// Mitsubishi GX Works2 project: Lycoming6p   PLC: FX3U/FX3UC
// AMX-FX3U with EM3A-AM8

PROGRAM MAIN
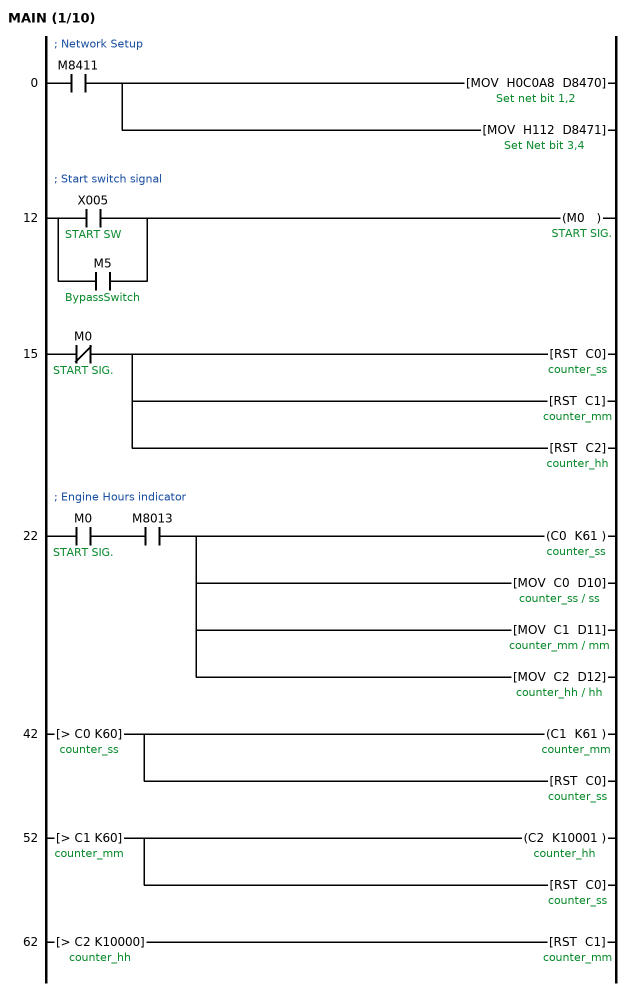
; Network Setup
0     LD      M8411
      MOV     H0C0A8 D8470  ; Set net bit 1,2
      MOV     H112 D8471  ; Set Net bit 3,4
; Start switch signal
12    LD      X005  ; START SW
      OR      M5  ; BypassSwitch
      OUT     M0  ; START SIG.
15    LDI     M0  ; START SIG.
      RST     C0  ; counter_ss
      RST     C1  ; counter_mm
      RST     C2  ; counter_hh
; Engine Hours indicator
22    LD      M0  ; START SIG.
      AND     M8013
      OUT     C0 K61  ; counter_ss
      MOV     C0 D10  ; ss
      MOV     C1 D11  ; mm
      MOV     C2 D12  ; hh
42    LD>     C0 K60  ; counter_ss
      OUT     C1 K61  ; counter_mm
      RST     C0  ; counter_ss
52    LD>     C1 K60  ; counter_mm
      OUT     C2 K10001  ; counter_hh
      RST     C0  ; counter_ss
62    LD>     C2 K10000  ; counter_hh
      RST     C1  ; counter_mm
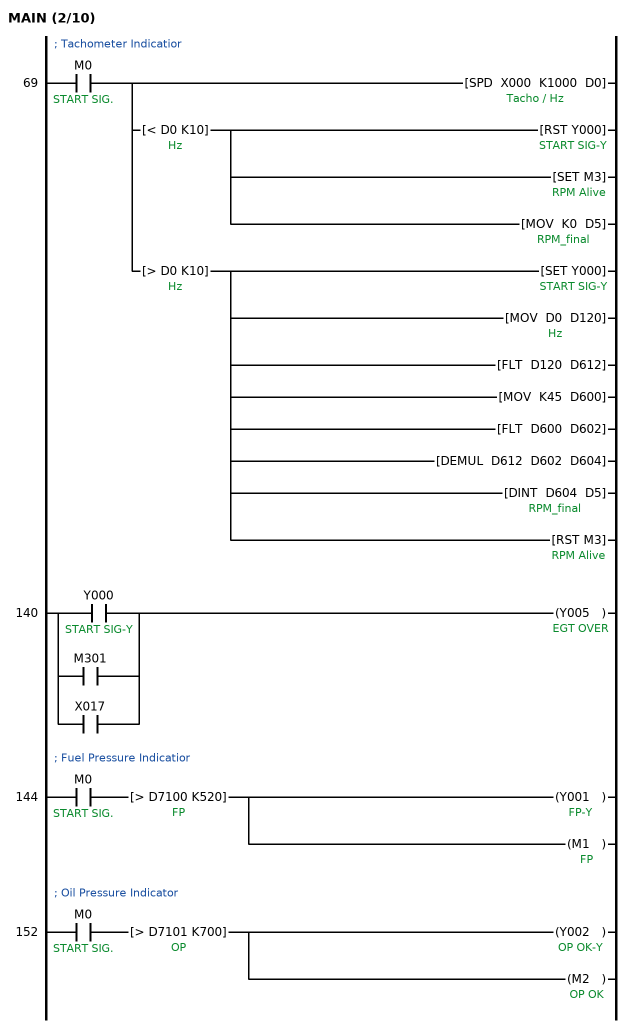
; Tachometer Indicatior
69    LD      M0  ; START SIG.
      SPD     X000 K1000 D0  ; Tacho / Hz
      MPS
      AND<    D0 K10  ; Hz
      RST     Y000  ; START SIG-Y
      SET     M3  ; RPM Alive
      MOV     K0 D5  ; RPM_final
      MPP
      AND>    D0 K10  ; Hz
      SET     Y000  ; START SIG-Y
      MOV     D0 D120
      FLT     D120 D612
      MOV     K45 D600
      FLT     D600 D602
      DEMUL   D612 D602 D604
      DINT    D604 D5
      RST     M3  ; RPM Alive
140   LD      Y000  ; START SIG-Y
      OR      M301
      OR      X017
      OUT     Y005  ; EGT OVER
; Fuel Pressure Indicatior
144   LD      M0  ; START SIG.
      AND>    D7100 K520  ; FP
      OUT     Y001  ; FP-Y
      OUT     M1  ; FP
; Oil Pressure Indicator
152   LD      M0  ; START SIG.
      AND>    D7101 K700  ; OP
      OUT     Y002  ; OP OK-Y
      OUT     M2  ; OP OK
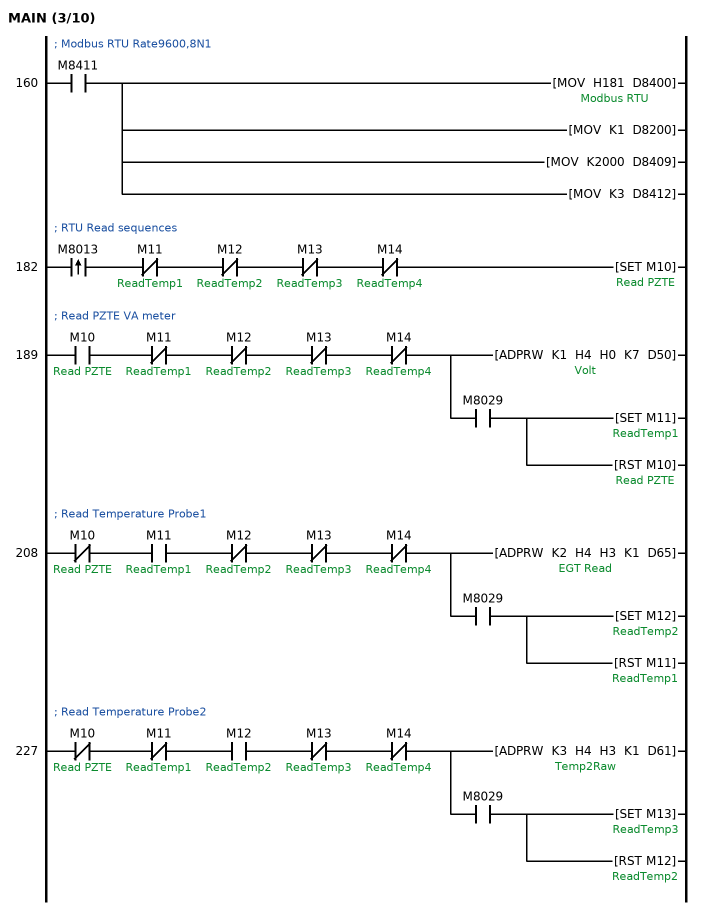
; Modbus RTU Rate9600,8N1
160   LD      M8411
      MOV     H181 D8400  ; Modbus RTU
      MOV     K1 D8200
      MOV     K2000 D8409
      MOV     K3 D8412
; RTU Read sequences
182   LDP     M8013
      ANI     M11  ; ReadTemp1
      ANI     M12  ; ReadTemp2
      ANI     M13  ; ReadTemp3
      ANI     M14  ; ReadTemp4
      SET     M10  ; Read PZTE
; Read PZTE VA meter
189   LD      M10  ; Read PZTE
      ANI     M11  ; ReadTemp1
      ANI     M12  ; ReadTemp2
      ANI     M13  ; ReadTemp3
      ANI     M14  ; ReadTemp4
      ADPRW   K1 H4 H0 K7 D50  ; Volt
      AND     M8029
      SET     M11  ; ReadTemp1
      RST     M10  ; Read PZTE
; Read Temperature Probe1
208   LDI     M10  ; Read PZTE
      AND     M11  ; ReadTemp1
      ANI     M12  ; ReadTemp2
      ANI     M13  ; ReadTemp3
      ANI     M14  ; ReadTemp4
      ADPRW   K2 H4 H3 K1 D65  ; EGT Read
      AND     M8029
      SET     M12  ; ReadTemp2
      RST     M11  ; ReadTemp1
; Read Temperature Probe2
227   LDI     M10  ; Read PZTE
      ANI     M11  ; ReadTemp1
      AND     M12  ; ReadTemp2
      ANI     M13  ; ReadTemp3
      ANI     M14  ; ReadTemp4
      ADPRW   K3 H4 H3 K1 D61  ; Temp2Raw
      AND     M8029
      SET     M13  ; ReadTemp3
      RST     M12  ; ReadTemp2
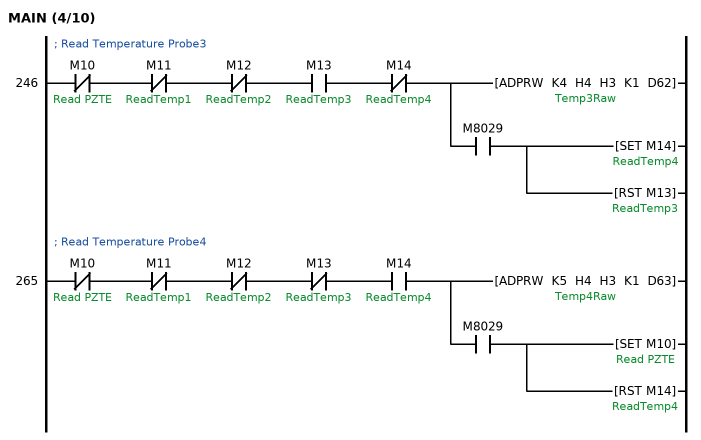
; Read Temperature Probe3
246   LDI     M10  ; Read PZTE
      ANI     M11  ; ReadTemp1
      ANI     M12  ; ReadTemp2
      AND     M13  ; ReadTemp3
      ANI     M14  ; ReadTemp4
      ADPRW   K4 H4 H3 K1 D62  ; Temp3Raw
      AND     M8029
      SET     M14  ; ReadTemp4
      RST     M13  ; ReadTemp3
; Read Temperature Probe4
265   LDI     M10  ; Read PZTE
      ANI     M11  ; ReadTemp1
      ANI     M12  ; ReadTemp2
      ANI     M13  ; ReadTemp3
      AND     M14  ; ReadTemp4
      ADPRW   K5 H4 H3 K1 D63  ; Temp4Raw
      AND     M8029
      SET     M10  ; Read PZTE
      RST     M14  ; ReadTemp4
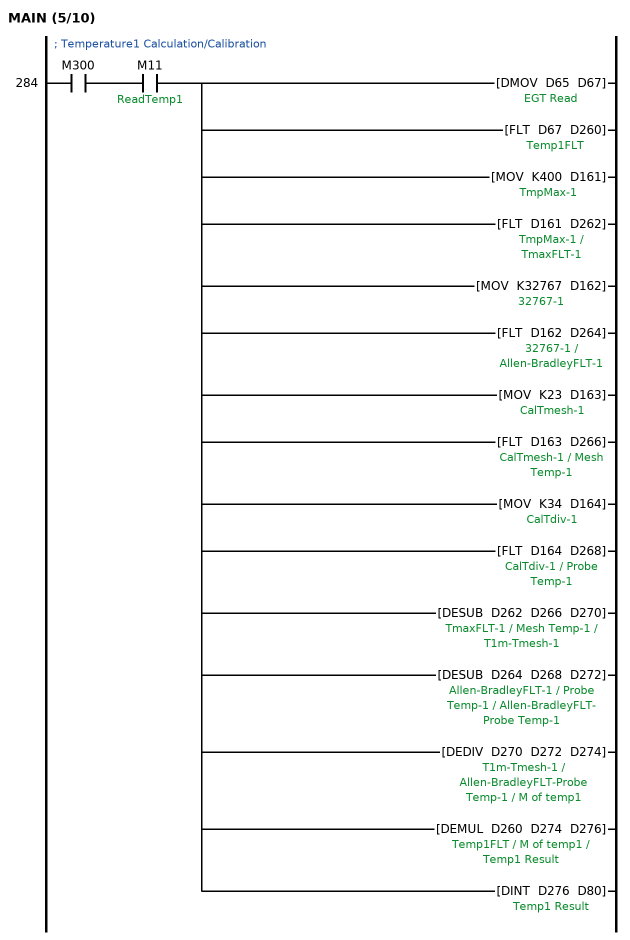
; Temperature1 Calculation/Calibration
284   LD      M300
      AND     M11  ; ReadTemp1
      DMOV    D65 D67
      FLT     D67 D260  ; Temp1FLT
      MOV     K400 D161  ; TmpMax-1
      FLT     D161 D262  ; TmaxFLT-1
      MOV     K32767 D162  ; 32767-1
      FLT     D162 D264  ; Allen-BradleyFLT-1
      MOV     K23 D163  ; CalTmesh-1
      FLT     D163 D266  ; Mesh Temp-1
      MOV     K34 D164  ; CalTdiv-1
      FLT     D164 D268  ; Probe Temp-1
      DESUB   D262 D266 D270  ; T1m-Tmesh-1
      DESUB   D264 D268 D272  ; Allen-BradleyFLT-Probe Temp-1
      DEDIV   D270 D272 D274  ; M of temp1
      DEMUL   D260 D274 D276  ; Temp1 Result
      DINT    D276 D80
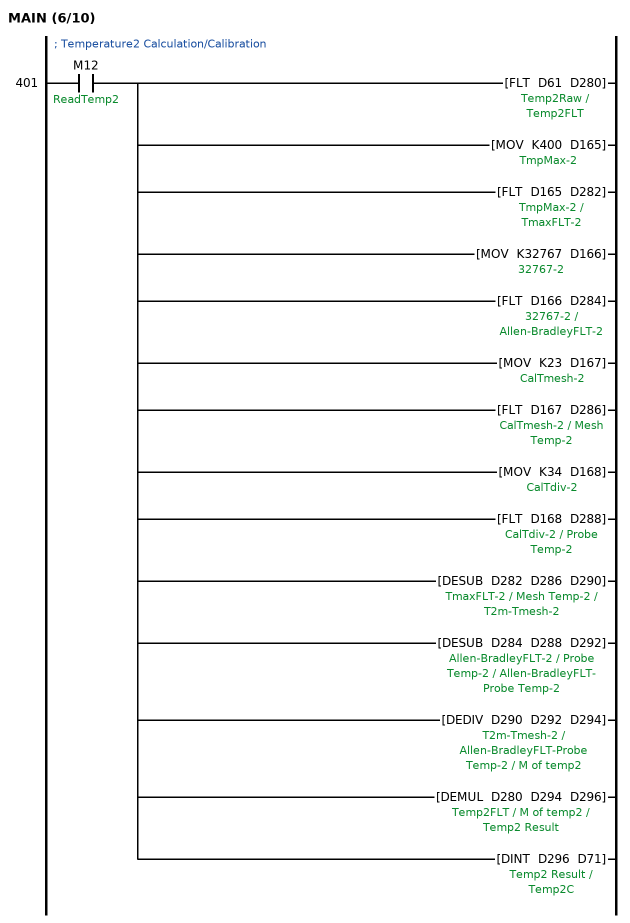
; Temperature2 Calculation/Calibration
401   LD      M12  ; ReadTemp2
      FLT     D61 D280  ; Temp2FLT
      MOV     K400 D165  ; TmpMax-2
      FLT     D165 D282  ; TmaxFLT-2
      MOV     K32767 D166  ; 32767-2
      FLT     D166 D284  ; Allen-BradleyFLT-2
      MOV     K23 D167  ; CalTmesh-2
      FLT     D167 D286  ; Mesh Temp-2
      MOV     K34 D168  ; CalTdiv-2
      FLT     D168 D288  ; Probe Temp-2
      DESUB   D282 D286 D290  ; T2m-Tmesh-2
      DESUB   D284 D288 D292  ; Allen-BradleyFLT-Probe Temp-2
      DEDIV   D290 D292 D294  ; M of temp2
      DEMUL   D280 D294 D296  ; Temp2 Result
      DINT    D296 D71  ; Temp2C
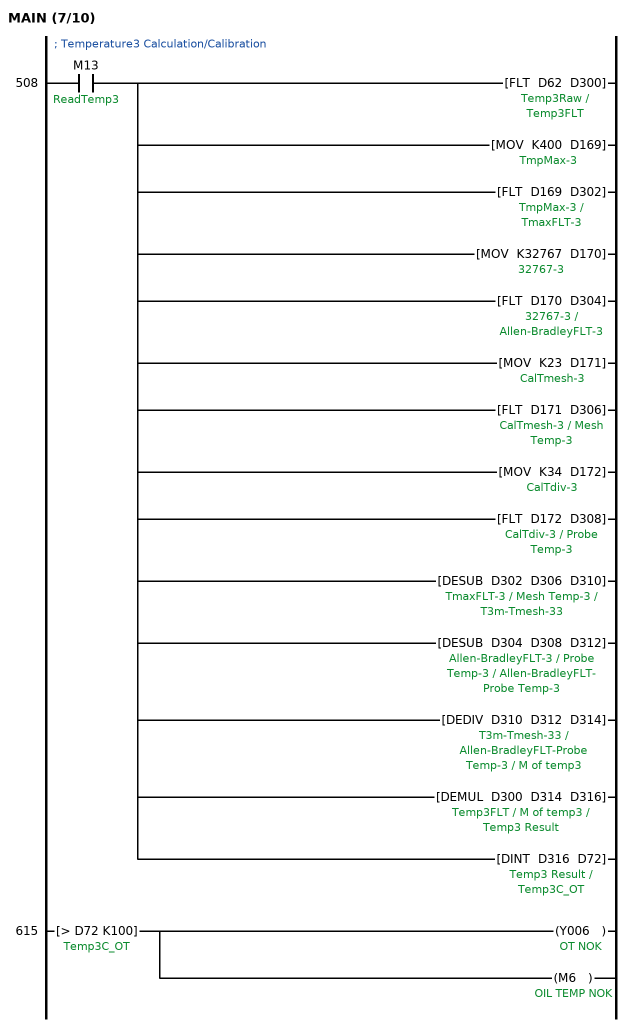
; Temperature3 Calculation/Calibration
508   LD      M13  ; ReadTemp3
      FLT     D62 D300  ; Temp3FLT
      MOV     K400 D169  ; TmpMax-3
      FLT     D169 D302  ; TmaxFLT-3
      MOV     K32767 D170  ; 32767-3
      FLT     D170 D304  ; Allen-BradleyFLT-3
      MOV     K23 D171  ; CalTmesh-3
      FLT     D171 D306  ; Mesh Temp-3
      MOV     K34 D172  ; CalTdiv-3
      FLT     D172 D308  ; Probe Temp-3
      DESUB   D302 D306 D310  ; T3m-Tmesh-33
      DESUB   D304 D308 D312  ; Allen-BradleyFLT-Probe Temp-3
      DEDIV   D310 D312 D314  ; M of temp3
      DEMUL   D300 D314 D316  ; Temp3 Result
      DINT    D316 D72  ; Temp3C_OT
615   LD>     D72 K100  ; Temp3C_OT
      OUT     Y006  ; OT NOK
      OUT     M6  ; OIL TEMP NOK
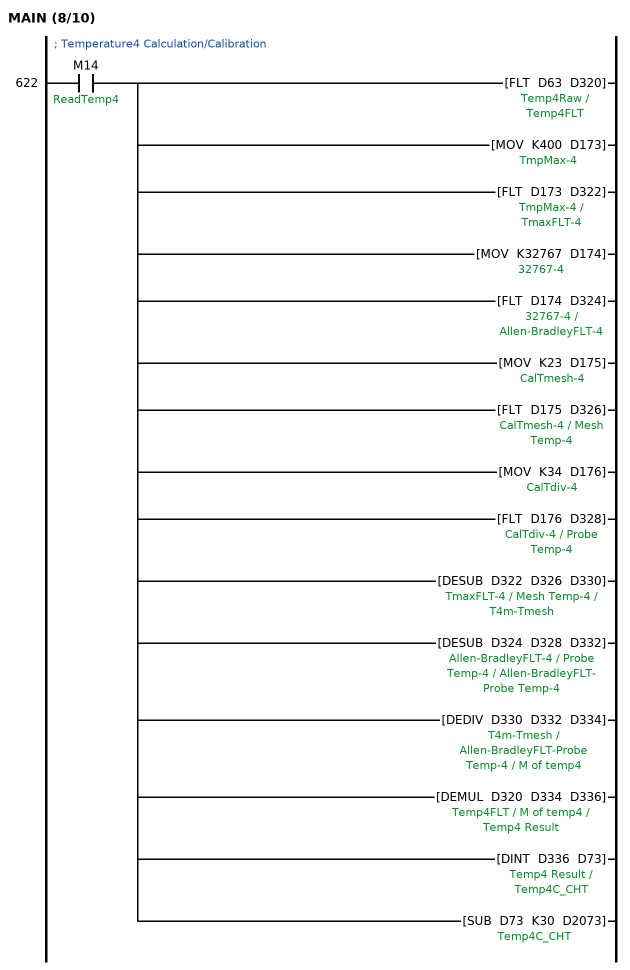
; Temperature4 Calculation/Calibration
622   LD      M14  ; ReadTemp4
      FLT     D63 D320  ; Temp4FLT
      MOV     K400 D173  ; TmpMax-4
      FLT     D173 D322  ; TmaxFLT-4
      MOV     K32767 D174  ; 32767-4
      FLT     D174 D324  ; Allen-BradleyFLT-4
      MOV     K23 D175  ; CalTmesh-4
      FLT     D175 D326  ; Mesh Temp-4
      MOV     K34 D176  ; CalTdiv-4
      FLT     D176 D328  ; Probe Temp-4
      DESUB   D322 D326 D330  ; T4m-Tmesh
      DESUB   D324 D328 D332  ; Allen-BradleyFLT-Probe Temp-4
      DEDIV   D330 D332 D334  ; M of temp4
      DEMUL   D320 D334 D336  ; Temp4 Result
      DINT    D336 D73  ; Temp4C_CHT
      SUB     D73 K30 D2073
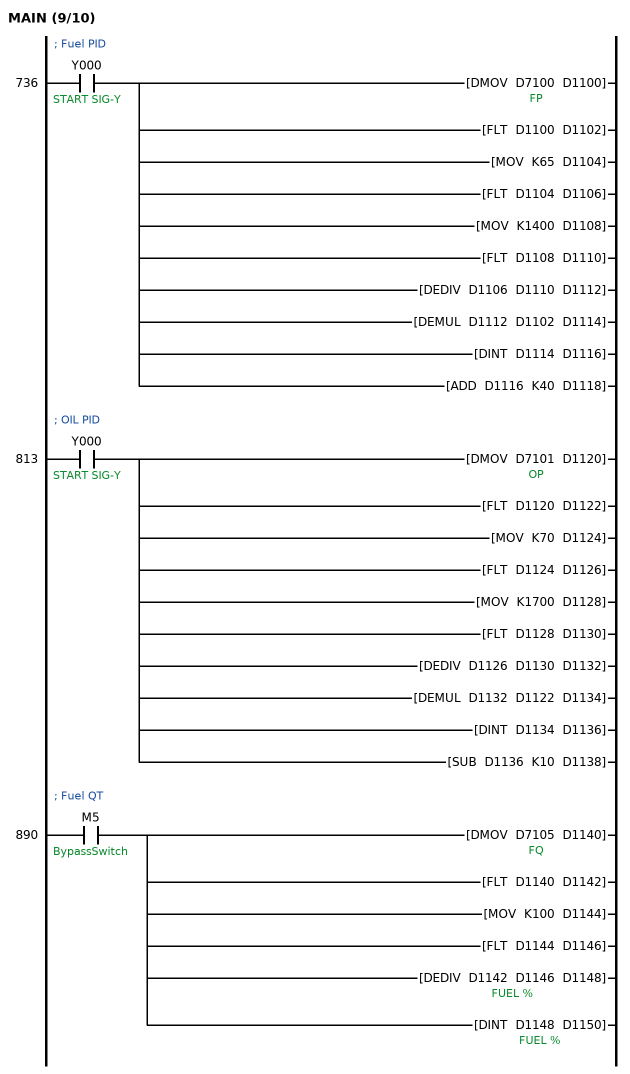
; Fuel PID
736   LD      Y000  ; START SIG-Y
      DMOV    D7100 D1100
      FLT     D1100 D1102
      MOV     K65 D1104
      FLT     D1104 D1106
      MOV     K1400 D1108
      FLT     D1108 D1110
      DEDIV   D1106 D1110 D1112
      DEMUL   D1112 D1102 D1114
      DINT    D1114 D1116
      ADD     D1116 K40 D1118
; OIL PID
813   LD      Y000  ; START SIG-Y
      DMOV    D7101 D1120
      FLT     D1120 D1122
      MOV     K70 D1124
      FLT     D1124 D1126
      MOV     K1700 D1128
      FLT     D1128 D1130
      DEDIV   D1126 D1130 D1132
      DEMUL   D1132 D1122 D1134
      DINT    D1134 D1136
      SUB     D1136 K10 D1138
; Fuel QT
890   LD      M5  ; BypassSwitch
      DMOV    D7105 D1140  ; FQ
      FLT     D1140 D1142
      MOV     K100 D1144
      FLT     D1144 D1146
      DEDIV   D1142 D1146 D1148  ; FUEL %
      DINT    D1148 D1150
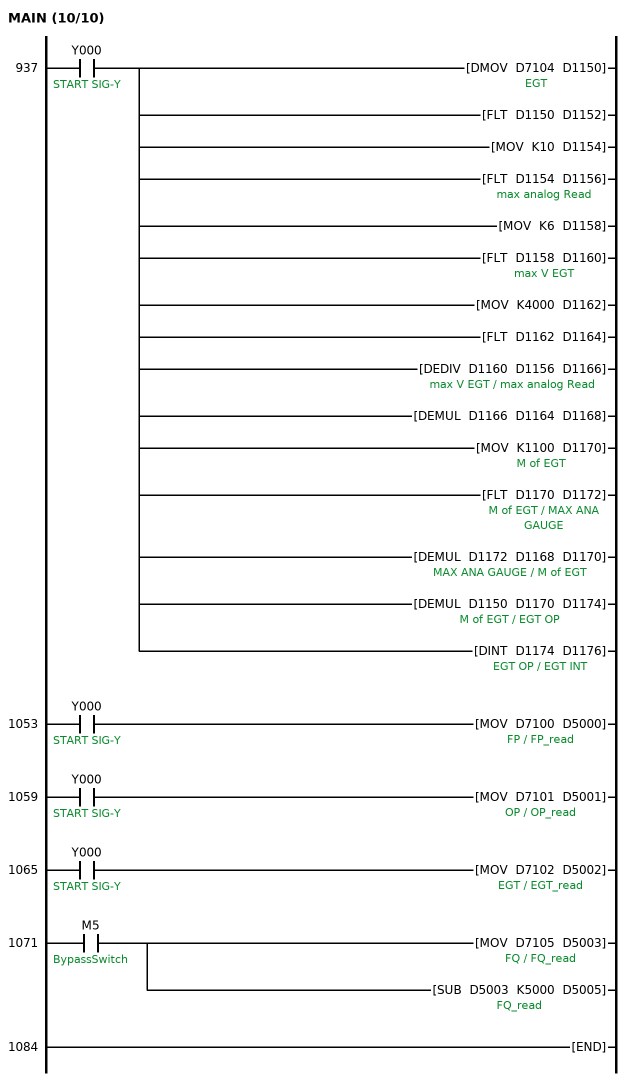
937   LD      Y000  ; START SIG-Y
      DMOV    D7104 D1150  ; EGT
      FLT     D1150 D1152
      MOV     K10 D1154
      FLT     D1154 D1156  ; max analog Read
      MOV     K6 D1158
      FLT     D1158 D1160  ; max V EGT
      MOV     K4000 D1162
      FLT     D1162 D1164
      DEDIV   D1160 D1156 D1166
      DEMUL   D1166 D1164 D1168
      MOV     K1100 D1170  ; M of EGT
      FLT     D1170 D1172  ; MAX ANA GAUGE
      DEMUL   D1172 D1168 D1170
      DEMUL   D1150 D1170 D1174  ; EGT OP
      DINT    D1174 D1176  ; EGT INT
1053  LD      Y000  ; START SIG-Y
      MOV     D7100 D5000  ; FP_read
1059  LD      Y000  ; START SIG-Y
      MOV     D7101 D5001  ; OP_read
1065  LD      Y000  ; START SIG-Y
      MOV     D7102 D5002  ; EGT / EGT_read
1071  LD      M5  ; BypassSwitch
      MOV     D7105 D5003  ; FQ_read
      SUB     D5003 K5000 D5005
1084  END
END_PROGRAM

// device comments not shown above
D1  ; RPM_cal
D2  ; RPM_show
D51  ; Amp
D52  ; F.Watt1
D53  ; F.Watt2
D54  ; Wh1
D55  ; Wh2
D56  ; AlarmH
D57  ; AlarmL
D60  ; Temp1Raw
D70  ; Temp1C
D7400  ; AM 8 OUTPUT1
D7401  ; AM 8 OUTPUT2
D7402  ; AM 8 OUTPUT3
D7403  ; AM 8 OUTPUT4
M4  ; Vaccum
Y003  ; RPM Alive-Y
Y004  ; Vaccum-Y
